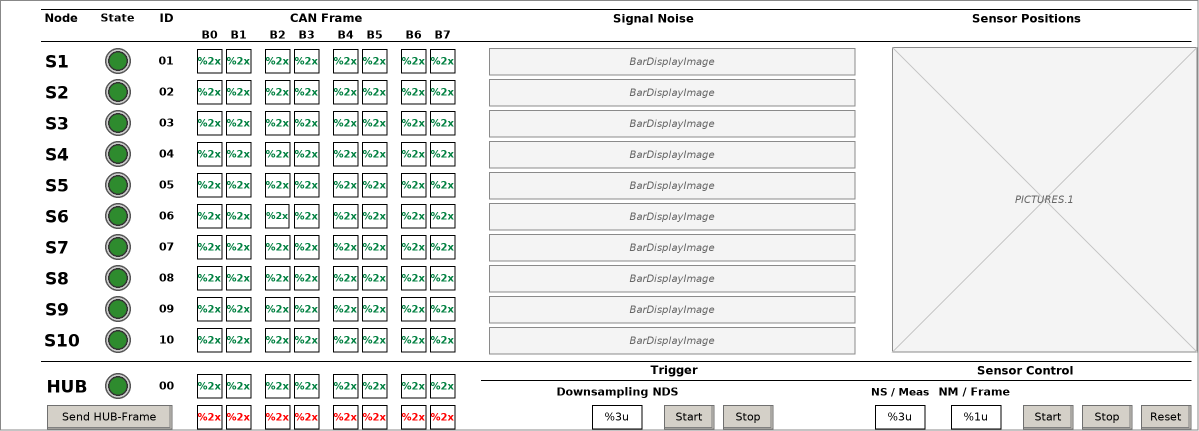
VISUALIZATION VISUALISATION_SENSOR_CONTROL  // 1199x431
    Group (870,363 321x66)
        Rectangle (65,17 79x24), "NM / Frame"
        Rectangle (0,17 61x24), "NS / Meas"
        Button (153,42 50x24), "Start"
            OnMouseClick: execute { CAN_CONTROL_STATE:=1; }
        Button (212,42 50x24), "Stop"
            OnMouseClick: execute { CAN_CONTROL_STATE:=0; }
        Button (271,42 50x24), "Reset"
            OnMouseClick: execute { CAN_CONTROL_STATE:=2; }
        Rectangle (81,42 50x24), "%1u", text variable: VARIABLES.M_PER_FRAME
            OnMouseDown: write the text variable via Default, min 0, max 4
        Rectangle (97,0 117x15), "Sensor Control"
        Rectangle (5,42 50x24), "%3u", text variable: VARIABLES.N_SAMPLES_PER_M
            OnMouseDown: write the text variable via Default, min 0, max 255
    Group (507,359 266x70)
        Rectangle (97,0 140x22), "Trigger"
        Button (157,46 50x24), "Start"
            OnMouseClick: execute { VARIABLES.CAN_TRIGGER_STATE:=1; }
        Rectangle (0,21 221x24), "Downsampling NDS"
        Rectangle (85,46 50x24), "%3u", text variable: VARIABLES.K_TRIGGER
            OnMouseDown: write the text variable via Default
        Button (216,46 50x24), "Stop"
            OnMouseClick: execute { VARIABLES.CAN_TRIGGER_STATE:=0; }
    Group (489,11 366x343)
        BarDisplayImage (0,37 366x27), value: VARIABLES.SIGNAL_DEVIATION[1], style: BarDisplayImage-Gray, scale format: %1u, scale 0..200
        BarDisplayImage (0,68 366x27), value: VARIABLES.SIGNAL_DEVIATION[2], style: BarDisplayImage-Gray, scale format: %1u, scale 0..200
        BarDisplayImage (0,99 366x27), value: VARIABLES.SIGNAL_DEVIATION[3], style: BarDisplayImage-Gray, scale format: %1u, scale 0..200
        BarDisplayImage (0,130 366x27), value: VARIABLES.SIGNAL_DEVIATION[4], style: BarDisplayImage-Gray, scale format: %1u, scale 0..200
        BarDisplayImage (0,161 366x27), value: VARIABLES.SIGNAL_DEVIATION[5], style: BarDisplayImage-Gray, scale format: %1u, scale 0..200
        BarDisplayImage (0,192 366x27), value: VARIABLES.SIGNAL_DEVIATION[6], style: BarDisplayImage-Gray, scale format: %1u, scale 0..200
        BarDisplayImage (0,223 366x27), value: VARIABLES.SIGNAL_DEVIATION[7], style: BarDisplayImage-Gray, scale format: %1u, scale 0..200
        Rectangle (106,0 117x15), "Signal Noise"
        BarDisplayImage (0,254 366x27), value: VARIABLES.SIGNAL_DEVIATION[8], style: BarDisplayImage-Gray, scale format: %1u, scale 0..200
        BarDisplayImage (0,285 366x27), value: VARIABLES.SIGNAL_DEVIATION[9], style: BarDisplayImage-Gray, scale format: %1u, scale 0..200
        BarDisplayImage (0,316 366x27), value: VARIABLES.SIGNAL_DEVIATION[10], style: BarDisplayImage-Gray, scale format: %1u, scale 0..200
    Group (29,371 426x58)
        Button (18,34 125x24), "Send HUB-Frame"
            OnMouseClick: execute { CAN_CONTROL_STATE:=3; }
        Rectangle (401,34 25x24), "%2x", text variable: VARIABLES.CAN_PARAMETER_FRAME[7]
            OnMouseDown: write the text variable via Default
        Rectangle (372,34 25x24), "%2x", text variable: VARIABLES.CAN_PARAMETER_FRAME[6]
            OnMouseDown: write the text variable via Default
        Rectangle (333,34 25x24), "%2x", text variable: VARIABLES.CAN_PARAMETER_FRAME[5]
            OnMouseDown: write the text variable via Default
        Rectangle (304,34 25x24), "%2x", text variable: VARIABLES.CAN_PARAMETER_FRAME[4]
            OnMouseDown: write the text variable via Default
        Rectangle (265,34 25x24), "%2x", text variable: VARIABLES.CAN_PARAMETER_FRAME[3]
            OnMouseDown: write the text variable via Default
        Rectangle (236,34 25x24), "%2x", text variable: VARIABLES.CAN_PARAMETER_FRAME[2]
            OnMouseDown: write the text variable via Default
        Rectangle (197,34 25x24), "%2x", text variable: VARIABLES.CAN_PARAMETER_FRAME[1]
            OnMouseDown: write the text variable via Default
        Rectangle (168,34 25x24), "%2x", text variable: VARIABLES.CAN_PARAMETER_FRAME[0]
            OnMouseDown: write the text variable via Default
        Rectangle (0,2 76x27), "HUB"
        Lamp1 (74,0 30x30), variable: VARIABLES.HUB_STATE, style: Lamp-Lamp1-Green
        Rectangle (168,3 25x24), "%2x", text variable: VARIABLES.CAN_HUB [0]
        Rectangle (197,3 25x24), "%2x", text variable: VARIABLES.CAN_HUB [1]
        Rectangle (236,3 25x24), "%2x", text variable: VARIABLES.CAN_HUB [2]
        Rectangle (265,3 25x24), "%2x", text variable: VARIABLES.CAN_HUB [3]
        Rectangle (304,3 25x24), "%2x", text variable: VARIABLES.CAN_HUB [4]
        Rectangle (333,3 25x24), "%2x", text variable: VARIABLES.CAN_HUB [5]
        Rectangle (372,3 25x24), "%2x", text variable: VARIABLES.CAN_HUB [6]
        Rectangle (401,3 25x24), "%2x", text variable: VARIABLES.CAN_HUB [7]
        Rectangle (125,3 25x24), "00"
    Group (19,13 436x342)
        Rectangle (0,35 76x27), "S1"
        Rectangle (0,66 76x27), "S2"
        Rectangle (0,97 76x27), "S3"
        Rectangle (0,128 76x27), "S4"
        Rectangle (0,159 76x27), "S5"
        Rectangle (0,190 76x27), "S6"
        Rectangle (0,221 76x27), "S7"
        Rectangle (0,252 76x27), "S8"
        Rectangle (0,283 76x27), "S9"
        Lamp1 (84,33 30x30), variable: VARIABLES.SENSOR_STATE[1], style: Lamp-Lamp1-Green
        Lamp1 (84,64 30x30), variable: VARIABLES.SENSOR_STATE[2], style: Lamp-Lamp1-Green
        Lamp1 (84,95 30x30), variable: VARIABLES.SENSOR_STATE[3], style: Lamp-Lamp1-Green
        Lamp1 (84,126 30x30), variable: VARIABLES.SENSOR_STATE[4], style: Lamp-Lamp1-Green
        Lamp1 (84,157 30x30), variable: VARIABLES.SENSOR_STATE[5], style: Lamp-Lamp1-Green
        Lamp1 (84,188 30x30), variable: VARIABLES.SENSOR_STATE[6], style: Lamp-Lamp1-Green
        Lamp1 (84,219 30x30), variable: VARIABLES.SENSOR_STATE[7], style: Lamp-Lamp1-Green
        Rectangle (178,10 25x24), "B0"
        Rectangle (207,10 25x24), "B1"
        Rectangle (246,10 25x24), "B2"
        Rectangle (275,10 25x24), "B3"
        Rectangle (314,10 25x24), "B4"
        Rectangle (343,10 25x24), "B5"
        Rectangle (382,10 25x24), "B6"
        Rectangle (411,10 25x24), "B7"
        Rectangle (270,0 75x10), "CAN Frame"
        Rectangle (130,0 35x10), "ID"
        Rectangle (18,0 49x10), "Node"
        Rectangle (81,0 35x10), "State"
        Lamp1 (84,250 30x30), variable: VARIABLES.SENSOR_STATE[8], style: Lamp-Lamp1-Green
        Lamp1 (84,281 30x30), variable: VARIABLES.SENSOR_STATE[9], style: Lamp-Lamp1-Green
        Rectangle (5,314 76x27), "S10"
        Lamp1 (84,312 30x30), variable: VARIABLES.SENSOR_STATE[10], style: Lamp-Lamp1-Green
        Rectangle (178,36 25x24), "%2x", text variable: VARIABLES.CAN_SENSOR_1 [0]
        Rectangle (207,36 25x24), "%2x", text variable: VARIABLES.CAN_SENSOR_1 [1]
        Rectangle (246,36 25x24), "%2x", text variable: VARIABLES.CAN_SENSOR_1 [2]
        Rectangle (275,36 25x24), "%2x", text variable: VARIABLES.CAN_SENSOR_1 [3]
        Rectangle (314,36 25x24), "%2x", text variable: VARIABLES.CAN_SENSOR_1 [4]
        Rectangle (343,36 25x24), "%2x", text variable: VARIABLES.CAN_SENSOR_1 [5]
        Rectangle (382,36 25x24), "%2x", text variable: VARIABLES.CAN_SENSOR_1 [6]
        Rectangle (411,36 25x24), "%2x", text variable: VARIABLES.CAN_SENSOR_1 [7]
        Rectangle (178,67 25x24), "%2x", text variable: VARIABLES.CAN_SENSOR_2 [0]
        Rectangle (207,67 25x24), "%2x", text variable: VARIABLES.CAN_SENSOR_2 [1]
        Rectangle (246,67 25x24), "%2x", text variable: VARIABLES.CAN_SENSOR_2 [2]
        Rectangle (275,67 25x24), "%2x", text variable: VARIABLES.CAN_SENSOR_2 [3]
        Rectangle (314,67 25x24), "%2x", text variable: VARIABLES.CAN_SENSOR_2 [4]
        Rectangle (343,67 25x24), "%2x", text variable: VARIABLES.CAN_SENSOR_2 [5]
        Rectangle (382,67 25x24), "%2x", text variable: VARIABLES.CAN_SENSOR_2 [6]
        Rectangle (411,67 25x24), "%2x", text variable: VARIABLES.CAN_SENSOR_2 [7]
        Rectangle (178,98 25x24), "%2x", text variable: VARIABLES.CAN_SENSOR_3 [0]
        Rectangle (207,98 25x24), "%2x", text variable: VARIABLES.CAN_SENSOR_3 [1]
        Rectangle (246,98 25x24), "%2x", text variable: VARIABLES.CAN_SENSOR_3 [2]
        Rectangle (275,98 25x24), "%2x", text variable: VARIABLES.CAN_SENSOR_3 [3]
        Rectangle (314,98 25x24), "%2x", text variable: VARIABLES.CAN_SENSOR_3 [4]
        Rectangle (343,98 25x24), "%2x", text variable: VARIABLES.CAN_SENSOR_3 [5]
        Rectangle (382,98 25x24), "%2x", text variable: VARIABLES.CAN_SENSOR_3 [6]
        Rectangle (411,98 25x24), "%2x", text variable: VARIABLES.CAN_SENSOR_3 [7]
        Rectangle (178,129 25x24), "%2x", text variable: VARIABLES.CAN_SENSOR_4 [0]
        Rectangle (207,129 25x24), "%2x", text variable: VARIABLES.CAN_SENSOR_4 [1]
        Rectangle (246,129 25x24), "%2x", text variable: VARIABLES.CAN_SENSOR_4 [2]
        Rectangle (275,129 25x24), "%2x", text variable: VARIABLES.CAN_SENSOR_4 [3]
        Rectangle (314,129 25x24), "%2x", text variable: VARIABLES.CAN_SENSOR_4 [4]
        Rectangle (343,129 25x24), "%2x", text variable: VARIABLES.CAN_SENSOR_4 [5]
        Rectangle (382,129 25x24), "%2x", text variable: VARIABLES.CAN_SENSOR_4 [6]
        Rectangle (411,129 25x24), "%2x", text variable: VARIABLES.CAN_SENSOR_4 [7]
        Rectangle (178,160 25x24), "%2x", text variable: VARIABLES.CAN_SENSOR_5 [0]
        Rectangle (207,160 25x24), "%2x", text variable: VARIABLES.CAN_SENSOR_5 [1]
        Rectangle (246,160 25x24), "%2x", text variable: VARIABLES.CAN_SENSOR_5 [2]
        Rectangle (275,160 25x24), "%2x", text variable: VARIABLES.CAN_SENSOR_5 [3]
        Rectangle (314,160 25x24), "%2x", text variable: VARIABLES.CAN_SENSOR_5 [4]
        Rectangle (343,160 25x24), "%2x", text variable: VARIABLES.CAN_SENSOR_5 [5]
        Rectangle (382,160 25x24), "%2x", text variable: VARIABLES.CAN_SENSOR_5 [6]
        Rectangle (411,160 25x24), "%2x", text variable: VARIABLES.CAN_SENSOR_5 [7]
        Rectangle (178,191 25x24), "%2x", text variable: VARIABLES.CAN_SENSOR_6[0]
        Rectangle (207,191 25x24), "%2x", text variable: VARIABLES.CAN_SENSOR_6[1]
        Rectangle (246,191 24x24), "%2x", text variable: VARIABLES.CAN_SENSOR_6 [2]
        Rectangle (275,191 25x24), "%2x", text variable: VARIABLES.CAN_SENSOR_6 [3]
        Rectangle (314,191 25x24), "%2x", text variable: VARIABLES.CAN_SENSOR_6[4]
        Rectangle (343,191 25x24), "%2x", text variable: VARIABLES.CAN_SENSOR_6 [5]
        Rectangle (382,191 25x24), "%2x", text variable: VARIABLES.CAN_SENSOR_6 [6]
        Rectangle (411,191 25x24), "%2x", text variable: VARIABLES.CAN_SENSOR_6[7]
        Rectangle (178,222 25x24), "%2x", text variable: VARIABLES.CAN_SENSOR_7 [0]
        Rectangle (207,222 25x24), "%2x", text variable: VARIABLES.CAN_SENSOR_7[1]
        Rectangle (246,222 25x24), "%2x", text variable: VARIABLES.CAN_SENSOR_7 [2]
        Rectangle (275,222 25x24), "%2x", text variable: VARIABLES.CAN_SENSOR_7 [3]
        Rectangle (314,222 25x24), "%2x", text variable: VARIABLES.CAN_SENSOR_7 [4]
        Rectangle (343,222 25x24), "%2x", text variable: VARIABLES.CAN_SENSOR_7 [5]
        Rectangle (382,222 25x24), "%2x", text variable: VARIABLES.CAN_SENSOR_7 [6]
        Rectangle (411,222 25x24), "%2x", text variable: VARIABLES.CAN_SENSOR_7 [7]
        Rectangle (135,36 24x24), "01"
        Rectangle (135,67 25x24), "02"
        Rectangle (135,98 25x24), "03"
        Rectangle (135,129 25x24), "04"
        Rectangle (135,160 25x24), "05"
        Rectangle (135,191 25x24), "1"
        Rectangle (135,191 25x24), "06"
        Rectangle (135,222 25x24), "07"
        Rectangle (178,253 25x24), "%2x", text variable: VARIABLES.CAN_SENSOR_8 [0]
        Rectangle (207,253 25x24), "%2x", text variable: VARIABLES.CAN_SENSOR_8[1]
        Rectangle (246,253 25x24), "%2x", text variable: VARIABLES.CAN_SENSOR_8 [2]
        Rectangle (275,253 25x24), "%2x", text variable: VARIABLES.CAN_SENSOR_8[3]
        Rectangle (314,253 25x24), "%2x", text variable: VARIABLES.CAN_SENSOR_8[4]
        Rectangle (343,253 25x24), "%2x", text variable: VARIABLES.CAN_SENSOR_8 [5]
        Rectangle (382,253 25x24), "%2x", text variable: VARIABLES.CAN_SENSOR_8 [6]
        Rectangle (411,253 25x24), "%2x", text variable: VARIABLES.CAN_SENSOR_8[7]
        Rectangle (178,284 25x24), "%2x", text variable: VARIABLES.CAN_SENSOR_9 [0]
        Rectangle (207,284 25x24), "%2x", text variable: VARIABLES.CAN_SENSOR_9 [1]
        Rectangle (246,284 25x24), "%2x", text variable: VARIABLES.CAN_SENSOR_9 [2]
        Rectangle (275,284 25x24), "%2x", text variable: VARIABLES.CAN_SENSOR_9 [3]
        Rectangle (314,284 25x24), "%2x", text variable: VARIABLES.CAN_SENSOR_9 [4]
        Rectangle (343,284 25x24), "%2x", text variable: VARIABLES.CAN_SENSOR_9 [5]
        Rectangle (382,284 25x24), "%2x", text variable: VARIABLES.CAN_SENSOR_9 [6]
        Rectangle (411,284 25x24), "%2x", text variable: VARIABLES.CAN_SENSOR_9 [7]
        Rectangle (178,315 25x24), "%2x", text variable: VARIABLES.CAN_SENSOR_10[0]
        Rectangle (207,315 25x24), "%2x", text variable: VARIABLES.CAN_SENSOR_10[1]
        Rectangle (246,315 25x24), "%2x", text variable: VARIABLES.CAN_SENSOR_10[2]
        Rectangle (275,315 25x24), "%2x", text variable: VARIABLES.CAN_SENSOR_10[3]
        Rectangle (314,315 25x24), "%2x", text variable: VARIABLES.CAN_SENSOR_10[4]
        Rectangle (343,315 25x24), "%2x", text variable: VARIABLES.CAN_SENSOR_10[5]
        Rectangle (382,315 25x24), "%2x", text variable: VARIABLES.CAN_SENSOR_10[6]
        Rectangle (411,315 25x24), "%2x", text variable: VARIABLES.CAN_SENSOR_10[7]
        Rectangle (135,253 25x24), "08"
        Rectangle (135,284 25x24), "1"
        Rectangle (135,284 25x24), "09"
        Rectangle (135,315 25x24), "10"
    Rectangle (968,11 117x15), "Sensor Positions"
    Image (892,47 305x305), image: PICTURES.1
    Line (41,9) (1191,9)
    Line (41,361) (1191,361)
    Line (481,380) (1191,380)
    Line (41,41) (1191,41)
END_VISUALIZATION

(* stored: Version 1.1.0.1, ProductVersion 3.1.0.26
   Visu VISUALISATION_SENSOR_CONTROL: Id {0c619658-6575-45d4-910d-10006ab29f77} *)
